// Mitsubishi GX Works2 project: semaforo   PLC: Q03UDV
// turma01

// task Task_01 (event TRUE, interval 0, priority 31): POU_01

PROGRAM POU_01
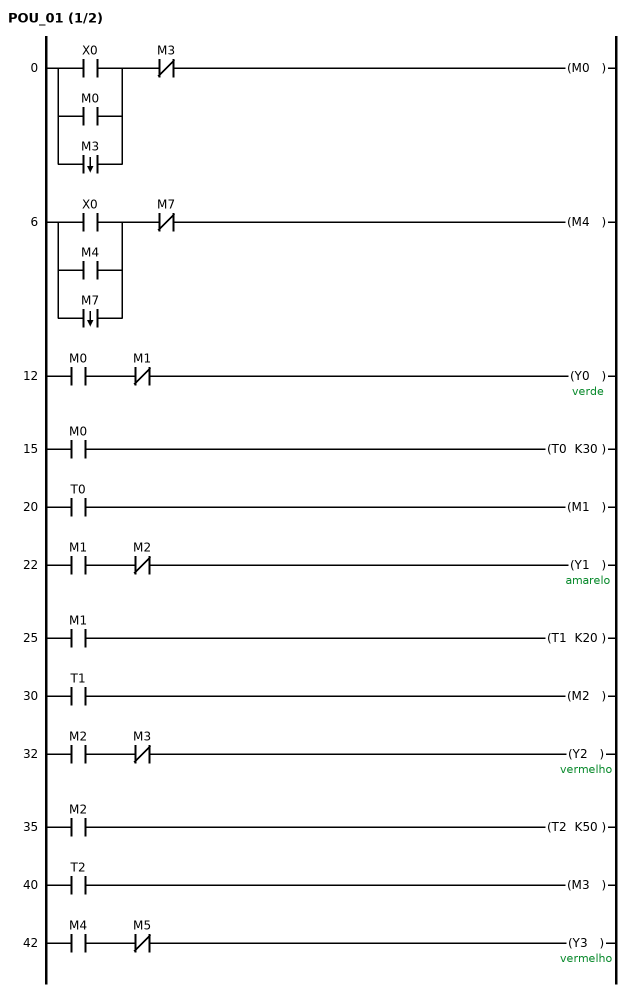
0     LD      X0
      OR      M0
      ORF     M3
      ANI     M3
      OUT     M0
6     LD      X0
      OR      M4
      ORF     M7
      ANI     M7
      OUT     M4
12    LD      M0
      ANI     M1
      OUT     Y0  ; verde
15    LD      M0
      OUT     T0 K30
20    LD      T0
      OUT     M1
22    LD      M1
      ANI     M2
      OUT     Y1  ; amarelo
25    LD      M1
      OUT     T1 K20
30    LD      T1
      OUT     M2
32    LD      M2
      ANI     M3
      OUT     Y2  ; vermelho
35    LD      M2
      OUT     T2 K50
40    LD      T2
      OUT     M3
42    LD      M4
      ANI     M5
      OUT     Y3  ; vermelho
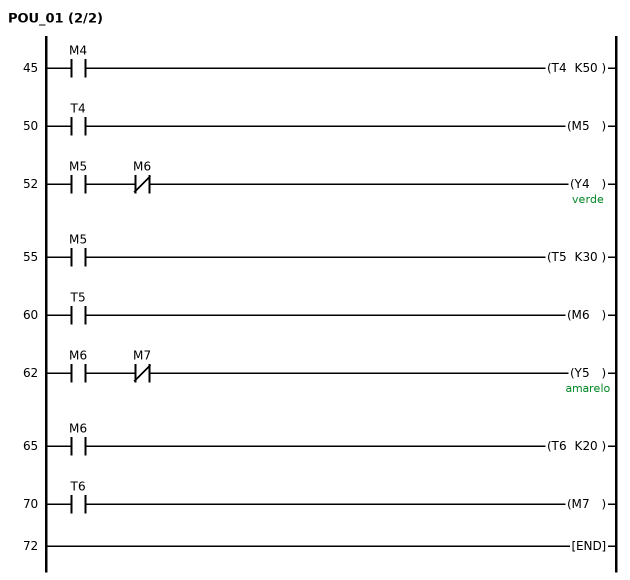
45    LD      M4
      OUT     T4 K50
50    LD      T4
      OUT     M5
52    LD      M5
      ANI     M6
      OUT     Y4  ; verde
55    LD      M5
      OUT     T5 K30
60    LD      T5
      OUT     M6
62    LD      M6
      ANI     M7
      OUT     Y5  ; amarelo
65    LD      M6
      OUT     T6 K20
70    LD      T6
      OUT     M7
72    END
END_PROGRAM
